// TIA Portal project "P3" (V20)

(* hardware
DEVICE "S7-1500/ET200MP station_1"  S7-1500 station
   slot 0: "Rail_0"  Rack  6ES7 590-1***0-0AA0
   slot 1: "PLC_1"  CPU 1511C-1 PN  6ES7 511-1CK01-0AB0  V2.9
      slot 3: "CPU display_1"  6ES7591-1AA00-0AA0
      slot 32768: "PROFINET interface_1"  X1
         slot 32769: "Port_1"  X1 P1
         slot 32770: "Port_2"  X1 P2
      slot 34817: "Virtual CP interface port_1"  Virtual CP interface port  Virtual CP interface port
*)

// ===== PLC "PLC_1"  CPU 1511C-1 PN =====

VAR_GLOBAL   // PLC tag table "Default tag table"
   "Tag_3" AT %Q1.0 : Bool;
   "Tag_4" AT %Q2.0 : Bool;
   "Tag_5" AT %Q3.0 : Bool;
   "Tag_2" AT %Q3.1 : Bool;
   "Tag_1" AT %Q0.1 : Bool;
   "ADD" AT %M0.1 : Bool;
   "Salida_EN0" AT %Q4.0 : Bool;
   "Suma" AT %M0.2 : Bool;
   "Salida_ADD" AT %Q5.0 : Bool;
END_VAR

DATA_BLOCK "Variables"   // DB1
{ S7_Optimized_Access := 'TRUE' }
VERSION : 0.1
   VAR
      Altura_Actual : Real := 5.0;
      Altura_Max : Real := 8.0;
      Altura_Min : Real := 2.0;
      Rango_Alto : Real := 6.0;
      Rango_Bajo : Real := 4.0;
      Res_1 : Real;
      Res_2 : Real;
      Res_3 : Real;
      Conversor : Real := 100.0;
      Salida : Real;
      Porcentaje : Real;
      Res_suma : Int;
   END_VAR
BEGIN
END_DATA_BLOCK

ORGANIZATION_BLOCK "Main"   // OB1, LAD, ProgramCycle
TITLE = "Main Program Sweep (Cycle)"
{ S7_Optimized_Access := 'TRUE' }
VERSION : 0.1
   VAR_INPUT
      Initial_Call : Bool;   // Initial call of this OB
      Remanence : Bool;   // =True, if remanent data are available
   END_VAR
BEGIN

REGION Network 1
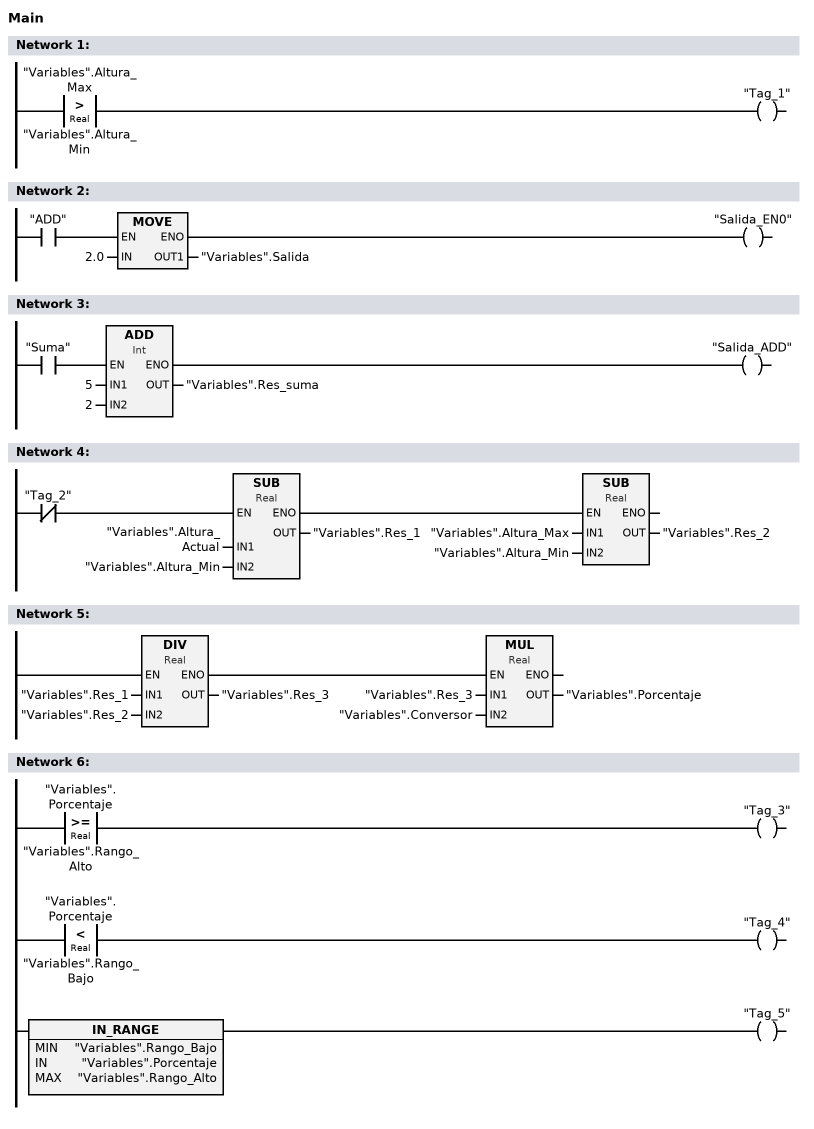
   RUNG wire#powerrail
      { S7_Templates := "SrcType := Real" } GT_Contact(in1 := "Variables".Altura_Max, in2 := "Variables".Altura_Min)
      Coil( "Tag_1" )
   END_RUNG
   // the same network as SCL:
   "Tag_1" := "Variables".Altura_Max > "Variables".Altura_Min;
END_REGION

REGION Network 2
   RUNG wire#powerrail
      Contact( "ADD" )
      Move(in := 2.0, out1 => "Variables".Salida)
      Coil( "Salida_EN0" )
   END_RUNG
   // the same network as SCL:
   IF "ADD" THEN "Variables".Salida := 2.0; END_IF;
   "Salida_EN0" := "ADD";
END_REGION

REGION Network 3
   RUNG wire#powerrail
      Contact( "Suma" )
      { S7_Templates := "SrcType := Int" } Add(in1 := 5, in2 := 2, out => "Variables".Res_suma)
      Coil( "Salida_ADD" )
   END_RUNG
   // the same network as SCL:
   IF "Suma" THEN "Variables".Res_suma := 5 + 2; END_IF;
   "Salida_ADD" := "Suma";
END_REGION

REGION Network 4
   RUNG wire#powerrail
      I_Contact( "Tag_2" )
      { S7_Templates := "SrcType := Real" } Sub(in1 := "Variables".Altura_Actual, in2 := "Variables".Altura_Min, out => "Variables".Res_1)
      { S7_Templates := "SrcType := Real" } Sub(in1 := "Variables".Altura_Max, in2 := "Variables".Altura_Min, out => "Variables".Res_2)
   END_RUNG
   // the same network as SCL:
   IF NOT "Tag_2" THEN
       "Variables".Res_1 := "Variables".Altura_Actual - "Variables".Altura_Min;
       "Variables".Res_2 := "Variables".Altura_Max - "Variables".Altura_Min;
   END_IF;
END_REGION

REGION Network 5
   RUNG wire#powerrail
      { S7_Templates := "SrcType := Real" } Div(in1 := "Variables".Res_1, in2 := "Variables".Res_2, out => "Variables".Res_3)
      { S7_Templates := "SrcType := Real" } Mul(in1 := "Variables".Res_3, in2 := "Variables".Conversor, out => "Variables".Porcentaje)
   END_RUNG
   // the same network as SCL:
   "Variables".Res_3 := "Variables".Res_1 / "Variables".Res_2;
   "Variables".Porcentaje := "Variables".Res_3 * "Variables".Conversor;
END_REGION

REGION Network 6
   RUNG wire#powerrail
      { S7_Templates := "SrcType := Real" } GE_Contact(in1 := "Variables".Porcentaje, in2 := "Variables".Rango_Alto)
      Coil( "Tag_3" )
   END_RUNG
   RUNG wire#powerrail
      { S7_Templates := "SrcType := Real" } LT_Contact(in1 := "Variables".Porcentaje, in2 := "Variables".Rango_Bajo)
      Coil( "Tag_4" )
   END_RUNG
   RUNG wire#powerrail
      { S7_Templates := "SrcType := Real" } InRange(min := "Variables".Rango_Bajo, in := "Variables".Porcentaje, max := "Variables".Rango_Alto)
      Coil( "Tag_5" )
   END_RUNG
   // the same network as SCL:
   "Tag_3" := "Variables".Porcentaje >= "Variables".Rango_Alto;
   "Tag_4" := "Variables".Porcentaje < "Variables".Rango_Bajo;
   "Tag_5" := ("Variables".Rango_Bajo <= "Variables".Porcentaje) AND ("Variables".Porcentaje <= "Variables".Rango_Alto);
END_REGION
END_ORGANIZATION_BLOCK